// TIA Portal V15.1 export
// export: Created 2024-06-21T08:40:42.8272233Z, ExportSetting WithDefaults, DisplayName Totally Integrated Automation Portal, DisplayVersion V15.1 Update 5, DisplayName TIA Portal Openness, DisplayVersion V15.1 Update 5, DisplayName SINAMICS Startdrive Advanced, DisplayVersion V15.1, DisplayName G130, G150, S120, S150, SINAMICS MV, S210, DisplayVersion V15.1, DisplayName G110M, G120, G120C, G120D, G120P, DisplayVersion V15.1, DisplayName STEP 7 Professional, DisplayVersion V15.1 Update 5, DisplayName STEP 7 Safety, DisplayVersion V15.1, DisplayName WinCC Professional, DisplayVersion V15.1 Update 5, DisplayName SIMATIC Visualization Architect, DisplayVersion V15.1
DATA_BLOCK "_DPComPLC212"   // DB261
{ S7_Optimized_Access := 'FALSE' }
AUTHOR : VCG
FAMILY : LocFncGn
NAME : 2011Intf
VERSION : 0.1
// stored: AutoNumber false, DBAccessibleFromOPCUA true, IsOnlyStoredInLoadMemory false, IsWriteProtectedInAS false
   VAR RETAIN
      AA_DPComCheckAlarm { ExternalAccessible := 'False'; ExternalVisible := 'False'; ExternalWritable := 'False'} : Bool;   // Alarm DP communication with PLC212 (LiveBit) / Alarm PN communication with PLCyyy (LiveBit)
      PLC212LDPCheckAlarmABCondition { ExternalAccessible := 'False'; ExternalVisible := 'False'; ExternalWritable := 'False'} : Bool;   // Alarm AB condition
      H_InBit0_15Anim : Word;   // Animation word for HMI
      H_TxtInBit0_15Anim : Struct   // Animation description of the bits
         "0" : String[50];   // Description
         "1" : String[50];   // Description
         "2" : String[50];   // Description
         "3" : String[50];   // Description
         "4" : String[50];   // Description
         "5" : String[50];   // Description
         "6" : String[50];   // Description
         "7" : String[50];   // Description
         "8" : String[50];   // Description
         "9" : String[50];   // Description
         "10" : String[50];   // Description
         "11" : String[50];   // Description
         "12" : String[50];   // Description
         "13" : String[50];   // Description
         "14" : String[50];   // Description
         "15" : String[50];   // Description
      END_STRUCT;
      H_InBit16_31Anim : Word;   // Animation word for HMI
      H_TxtInBit16_31Anim : Struct   // Animation description of the bits
         "0" : String[50];   // Description
         "1" : String[50];   // Description
         "2" : String[50];   // Description
         "3" : String[50];   // Description
         "4" : String[50];   // Description
         "5" : String[50];   // Description
         "6" : String[50];   // Description
         "7" : String[50];   // Description
         "8" : String[50];   // Description
         "9" : String[50];   // Description
         "10" : String[50];   // Description
         "11" : String[50];   // Description
         "12" : String[50];   // Description
         "13" : String[50];   // Description
         "14" : String[50];   // Description
         "15" : String[50];   // Description
      END_STRUCT;
      H_OutBit0_15Anim : Word;   // Animation word for HMI
      H_TxtOutBit0_15Anim : Struct   // Animation description of the bits
         "0" : String[50];   // Description
         "1" : String[50];   // Description
         "2" : String[50];   // Description
         "3" : String[50];   // Description
         "4" : String[50];   // Description
         "5" : String[50];   // Description
         "6" : String[50];   // Description
         "7" : String[50];   // Description
         "8" : String[50];   // Description
         "9" : String[50];   // Description
         "10" : String[50];   // Description
         "11" : String[50];   // Description
         "12" : String[50];   // Description
         "13" : String[50];   // Description
         "14" : String[50];   // Description
         "15" : String[50];   // Description
      END_STRUCT;
      H_OutBit16_31Anim : Word;   // Animation word for HMI
      H_TxtOutBit16_31Anim : Struct   // Animation description of the bits
         "0" : String[50];   // Description
         "1" : String[50];   // Description
         "2" : String[50];   // Description
         "3" : String[50];   // Description
         "4" : String[50];   // Description
         "5" : String[50];   // Description
         "6" : String[50];   // Description
         "7" : String[50];   // Description
         "8" : String[50];   // Description
         "9" : String[50];   // Description
         "10" : String[50];   // Description
         "11" : String[50];   // Description
         "12" : String[50];   // Description
         "13" : String[50];   // Description
         "14" : String[50];   // Description
         "15" : String[50];   // Description
      END_STRUCT;
      H_FInBit0_15Anim : Word;   // Animation word for HMI
      H_TxtFInBit0_15Anim : Struct   // Animation description of the bits
         "0" : String[50];   // Description
         "1" : String[50];   // Description
         "2" : String[50];   // Description
         "3" : String[50];   // Description
         "4" : String[50];   // Description
         "5" : String[50];   // Description
         "6" : String[50];   // Description
         "7" : String[50];   // Description
         "8" : String[50];   // Description
         "9" : String[50];   // Description
         "10" : String[50];   // Description
         "11" : String[50];   // Description
         "12" : String[50];   // Description
         "13" : String[50];   // Description
         "14" : String[50];   // Description
         "15" : String[50];   // Description
      END_STRUCT;
      H_FOutBit0_15Anim : Word;   // Animation word for HMI
      H_TxtFOutBit0_15Anim : Struct   // Animation description of the bits
         "0" : String[50];   // Description
         "1" : String[50];   // Description
         "2" : String[50];   // Description
         "3" : String[50];   // Description
         "4" : String[50];   // Description
         "5" : String[50];   // Description
         "6" : String[50];   // Description
         "7" : String[50];   // Description
         "8" : String[50];   // Description
         "9" : String[50];   // Description
         "10" : String[50];   // Description
         "11" : String[50];   // Description
         "12" : String[50];   // Description
         "13" : String[50];   // Description
         "14" : String[50];   // Description
         "15" : String[50];   // Description
      END_STRUCT;
      H_PLC212LDPCheckIAnim : Word;   // Animation word for HMI
      H_Anim : Word;   // Animation
      H_DBnr : Int;   // DB number
      H_HMICmd : Word;   // HMI command
      H_209210NCB02_BodyID : DInt;   // Animation Body ID Number
      H_209210NCB02_BodyTypeMatrix : DInt;   // Animation Body Type Matrix 7 digits
      H_209210NCB02_Routing : Int;   // Animation Routing Information
      H_209220NCB02_BodyID : DInt;   // Animation Body ID Number
      H_209220NCB02_BodyTypeMatrix : DInt;   // Animation Body Type Matrix 7 digits
      H_209220NCB02_Routing : Int;   // Animation Routing Information
      AlarmA { ExternalAccessible := 'False'; ExternalVisible := 'False'; ExternalWritable := 'False'} : Bool;   // Alarm A
      AlarmB { ExternalAccessible := 'False'; ExternalVisible := 'False'; ExternalWritable := 'False'} : Bool;   // Alarm B
      AlarmC { ExternalAccessible := 'False'; ExternalVisible := 'False'; ExternalWritable := 'False'} : Bool;   // Alarm C
      AlarmD { ExternalAccessible := 'False'; ExternalVisible := 'False'; ExternalWritable := 'False'} : Bool;   // Alarm D
      AlarmABCondition { ExternalAccessible := 'False'; ExternalVisible := 'False'; ExternalWritable := 'False'} : Bool;   // Alarm AB condition
      "______R228.01 --> 210CR23______" { ExternalAccessible := 'False'; ExternalVisible := 'False'; ExternalWritable := 'False'} : Bool;   // -----------------------------------------------------------------------------------
      "212AAccessStopRequest" { ExternalAccessible := 'False'; ExternalVisible := 'False'; ExternalWritable := 'False'} : Bool;   // Access Stop Request
      "212AS36/AS37ResetPB" { ExternalAccessible := 'False'; ExternalVisible := 'False'; ExternalWritable := 'False'} : Bool;   // AS Light Curtain - Push button Reset
      "212AS36/AS37StartPB" { ExternalAccessible := 'False'; ExternalVisible := 'False'; ExternalWritable := 'False'} : Bool;   // AS Light Curtain - Push button Start
      "212AS36/AS37StopPB" { ExternalAccessible := 'False'; ExternalVisible := 'False'; ExternalWritable := 'False'} : Bool;   // AS Light Curtain - Push button Stop
      "212AIAnim" { ExternalAccessible := 'False'; ExternalVisible := 'False'; ExternalWritable := 'False'} : Word;   // For animation of icon
      "212AModes" { ExternalAccessible := 'False'; ExternalVisible := 'False'; ExternalWritable := 'False'} : "Modes";   // Modes
      "R228.01" { ExternalAccessible := 'False'; ExternalVisible := 'False'; ExternalWritable := 'False'} : "Conveyor";   // Transfer
      "______R228.02 --> 220CR23______" { ExternalAccessible := 'False'; ExternalVisible := 'False'; ExternalWritable := 'False'} : Bool;   // -----------------------------------------------------------------------------------
      "212AS38/AS39ResetPB" { ExternalAccessible := 'False'; ExternalVisible := 'False'; ExternalWritable := 'False'} : Bool;   // AS Light Curtain - Push button Reset
      "212AS38/AS39StartPB" { ExternalAccessible := 'False'; ExternalVisible := 'False'; ExternalWritable := 'False'} : Bool;   // AS Light Curtain - Push button Start
      "212AS38/AS39StopPB" { ExternalAccessible := 'False'; ExternalVisible := 'False'; ExternalWritable := 'False'} : Bool;   // AS Light Curtain - Push button Stop
      "R228.02" { ExternalAccessible := 'False'; ExternalVisible := 'False'; ExternalWritable := 'False'} : "Conveyor";   // Transfer
      "______R230.03 --> 230CA21______" { ExternalAccessible := 'False'; ExternalVisible := 'False'; ExternalWritable := 'False'} : Bool;   // -----------------------------------------------------------------------------------
      "212AS40ResetPB" { ExternalAccessible := 'False'; ExternalVisible := 'False'; ExternalWritable := 'False'} : Bool;   // AS Light Curtain - Push button Reset
      "212AS40StartPB" { ExternalAccessible := 'False'; ExternalVisible := 'False'; ExternalWritable := 'False'} : Bool;   // AS Light Curtain - Push button Start
      "212AS40StopPB" { ExternalAccessible := 'False'; ExternalVisible := 'False'; ExternalWritable := 'False'} : Bool;   // AS Light Curtain - Push button Stop
      "212DIAnim" { ExternalAccessible := 'False'; ExternalVisible := 'False'; ExternalWritable := 'False'} : Word;   // For animation of icon
      "212DModes" { ExternalAccessible := 'False'; ExternalVisible := 'False'; ExternalWritable := 'False'} : "Modes";   // Modes
      "R230.03" { ExternalAccessible := 'False'; ExternalVisible := 'False'; ExternalWritable := 'False'} : "Conveyor";   // Transfer
      "R230.03SG9" { ExternalAccessible := 'False'; ExternalVisible := 'False'; ExternalWritable := 'False'} : Bool;   // Stop detection set
   END_VAR
BEGIN
END_DATA_BLOCK
